(* PLC project Tc2_System.F_ToCHR Demo, tc3-libraries-kb TwinCAT 3.1 *)
(* stored: creationDateTime 2026-05-20T00:00:00, modificationDateTime 2026-05-20T00:00:00 *)

PROGRAM P_Demo_F_ToCHR
  VAR
    byAsciiCode : BYTE := 16#31;  (* ASCII 码 0x31 = '1' *)
    sChar : STRING;  (* 转换得到的单字符字符串 *)
  END_VAR

// ============================================================
// Tc2_System.F_ToCHR 演示程序
// ============================================================
// 场景：通讯报文调试，把读到的字节流逐字节转 STRING 拼显示文本。
// 价值：替代手写 ASCII 转换表。
// 验证：登录后看 sChar = '1'。改 byAsciiCode 为 16#41 后 sChar 应变为 'A'；改为 16#0D（CR 回车）后 HMI 上可能只看到换行而看不到字符。
// 验证步骤：
//   1. 右键 PLC 项目 → Import PLCopenXML → 选本文件
//   2. 引用 Tc2_System（References → Add library）
//   3. 编译 → 登录 → 运行；按上方『验证』指引在线写值观察
// ============================================================

sChar := F_ToCHR(byAsciiCode);
END_PROGRAM
